FUNCTION_BLOCK FB_trocarCheckDetect
VAR_INPUT
END_VAR
VAR_OUTPUT
END_VAR
VAR
	m_trocarOnCounts :INT :=0;
	m_trocarOnCountThres :INT :=30;
END_VAR

METHOD run : BOOL
VAR_INPUT
	IOValue :UDINT;
END_VAR

VAR_OUTPUT
	
END_VAR
// torcar 
IF 32=(IOValue AND 16#20) THEN
	m_trocarOnCounts :=MIN(m_trocarOnCounts +1,m_trocarOnCountThres);
ELSE
	m_trocarOnCounts :=0;
END_IF

run := m_trocarOnCounts >= m_trocarOnCountThres;
END_METHOD

END_FUNCTION_BLOCK

(* stored: Version 1.1.0.1, ProductVersion 3.1.4024.11
   POU FB_trocarCheckDetect: Id {81d1bf0f-7c45-4b6a-a39e-cc9612e1a983}, SpecialFunc None
   Method run: Id {04823216-c21d-41ca-a38a-b90070268aed} *)
